FUNCTION_BLOCK FB_BaseControlElementDecoratorParent EXTENDS FB_BaseComponentDecoratorParent IMPLEMENTS ITF_BaseControlElementDecoratorParent
VAR
	itfControlElement				: ITF_BaseControlElement;
END_VAR

(*			
	EVERDE sp. z o.o.
	Rafał Osajda		24.03.2025		TC 4024.66
	Definicja nowego zgłoszenia
*)
METHOD PUBLIC EventsDefinition : BOOL
EventsDefinition		:= THIS^.itfControlElement.EventsDefinition ();
END_METHOD

(*			
	EVERDE sp. z o.o.
	Rafał Osajda		27.03.2025		TC 4024.66
	Obsluga bledow sprawdzanie czy jakis blad sie nei pojawil i ustawienie stanu lub wylaczenie
*)
METHOD PUBLIC ExecuteEveryCycle_Error
VAR_INPUT
END_VAR
THIS^.itfControlElement.ExecuteEveryCycle_Error ();
END_METHOD

(*			
	EVERDE sp. z o.o.
	Rafał Osajda		27.03.2025		TC 4024.66
	Wywolanie co cykl operacji 
*)
METHOD PUBLIC ExecuteEveryCycle_Operation
VAR_INPUT
END_VAR
THIS^.itfControlElement.ExecuteEveryCycle_Operation ();
END_METHOD

(*			
	EVERDE sp. z o.o.
	Rafał Osajda		27.03.2025		TC 4024.66
	Aktualizacja flag 
*)
METHOD PUBLIC ExecuteEveryCycle_Status
VAR_INST
END_VAR
THIS^.itfControlElement.ExecuteEveryCycle_Status ();
END_METHOD

(*			
	EVERDE sp. z o.o.
	Rafał Osajda		27.03.2025		TC 4024.66
	Testowanie czy nei pojawil sie jakis rozkaz i uruchomienie odpowiednich operacji
*)
METHOD PUBLIC ExecuteEveryCycle_Test
VAR_INPUT
END_VAR
THIS^.itfControlElement.ExecuteEveryCycle_Test ();
END_METHOD

METHOD FB_init : BOOL
VAR_INPUT
	bInitRetains : BOOL; // if TRUE, the retain variables are initialized (warm start / cold start)
	bInCopyCode : BOOL;  // if TRUE, the instance afterwards gets moved into the copy code (online change)
	fbToDecorate		: ITF_DecoratedElement;
END_VAR
THIS^.itfControlElement	:= fbToDecorate.GetITFControlElement ();
END_METHOD

(*			
	EVERDE sp. z o.o.
	Rafał Osajda		03.10.2025		TC 4024.66
	
*)
METHOD PUBLIC FirstCycle : BOOL
VAR_INPUT
END_VAR
FirstCycle				:= THIS^.itfControlElement.FirstCycle ();
END_METHOD

METHOD PUBLIC GetCode : STRING
VAR_INPUT
END_VAR
GetCode			:= THIS^.itfControlElement.GetCode ();
END_METHOD

(*			
	EVERDE sp. z o.o.
	Rafał Osajda		30.04.2025		TC 4024.66
	Zwraca czy element jest czymś zajety
*)
METHOD PUBLIC GetDoNothing : BOOL
GetDoNothing		:= THIS^.itfControlElement.GetDoNothing ();
END_METHOD

METHOD PUBLIC GetID : UINT
VAR_INPUT
END_VAR
GetID		:= THIS^.itfControlElement.GetID ();
END_METHOD

METHOD PUBLIC GetIdentyfier : ST_BaseElementIdentifier
VAR_INPUT
END_VAR
GetIdentyfier		:= THIS^.itfControlElement.GetIdentyfier ();
END_METHOD

METHOD PUBLIC GetName : ST_BaseLabel
VAR_INPUT
END_VAR
GetName		:= THIS^.itfControlElement.GetName ();
END_METHOD

(*			
	EVERDE sp. z o.o.
	Rafał Osajda		30.04.2025		TC 4024.66
	Zwraca czy element jest w pozycji 0 - referencyjnej
*)
METHOD PUBLIC GetPosition0 : BOOL
GetPosition0	:= THIS^.itfControlElement.GetPosition0 ();
END_METHOD

METHOD PUBLIC GetType : E_BaseElementType
VAR_INPUT
END_VAR
GetType		:= THIS^.itfControlElement.GetType ();
END_METHOD

(*			
	EVERDE sp. z o.o.
	Rafał Osajda		31.03.2025		TC 4024.66
	Flaga że w tej sesji pracy maszyny element został już wybazowany
*)
METHOD PUBLIC HomingGetDone : BOOL
VAR_INPUT
END_VAR
HomingGetDone	:= THIS^.itfControlElement.HomingGetDone ();
END_METHOD

(*			
	EVERDE sp. z o.o.
	Rafał Osajda		11.04.2025		TC 4024.66
	Zwraca czy bazowanie jest potrzebne
*)
METHOD PUBLIC HomingGetIsNeeded : BOOL
VAR_INPUT
END_VAR
HomingGetIsNeeded	:= THIS^.itfControlElement.HomingGetIsNeeded ();
END_METHOD

(*			
	EVERDE sp. z o.o.
	Rafał Osajda		27.05.2025		TC 4024.66
	Uruchomienie metody bazowania
*)
METHOD PUBLIC HomingStart
VAR_INPUT
END_VAR
THIS^.itfControlElement.HomingStart ();
END_METHOD

METHOD PUBLIC IsValidCommonData : BOOL
VAR_INPUT
END_VAR
IsValidCommonData			:= THIS^.itfControlElement.IsValidCommonData ();
END_METHOD

(*			
	EVERDE sp. z o.o.
	Rafał Osajda		07.10.2025		TC 4024.66
	Dodpisywanie się do listy logera
*)
METHOD PUBLIC JoinTheLogger : BOOL
VAR_INPUT
END_VAR
JoinTheLogger	:= THIS^.itfControlElement.JoinTheLogger ();
END_METHOD

METHOD PUBLIC LinkCommonData : BOOL
VAR_INPUT
	stCommonData				: REFERENCE TO ST_BaseCommonData;
END_VAR
LinkCommonData			:= THIS^.itfControlElement.LinkCommonData (stCommonData := stCommonData);
END_METHOD

METHOD PUBLIC LinkSS1 : BOOL
VAR_INPUT
	fbSS1			: ITF_BaseFlagGet;
END_VAR
LinkSS1		:= THIS^.itfControlElement.LinkSS1 (fbSS1 := fbSS1);
END_METHOD

METHOD PUBLIC LinkSTO : BOOL
VAR_INPUT
	fbSTO			: ITF_BaseFlagGet;
END_VAR
LinkSTO		:= THIS^.itfControlElement.LinkSTO (fbSTO := fbSTO);
END_METHOD

(*			
	EVERDE sp. z o.o.
	Rafał Osajda		31.03.2025		TC 4024.66
	Zwraca status zasilania	
*)
METHOD PUBLIC PowerGetStatus : BOOL
VAR_INPUT
END_VAR
PowerGetStatus		:= THIS^.itfControlElement.PowerGetStatus ();
END_METHOD

(*			
	EVERDE sp. z o.o.
	Rafał Osajda		31.03.2025		TC 4024.66
	Wyłączenie zasilania
*)
METHOD PUBLIC PowerTurnOff : BOOL
VAR_INPUT
END_VAR
PowerTurnOff		:= THIS^.itfControlElement.PowerTurnOff ();
END_METHOD

(*			
	EVERDE sp. z o.o.
	Rafał Osajda		31.03.2025		TC 4024.66
	Uruchomienie zasialania
*)
METHOD PUBLIC PowerTurnOn
VAR_INPUT
END_VAR
THIS^.itfControlElement.PowerTurnOn ();
END_METHOD

METHOD PUBLIC Reset : BOOL
VAR_INPUT
END_VAR
Reset	:= THIS^.itfControlElement.Reset ();
END_METHOD

METHOD PUBLIC ResetGetBusy : BOOL
VAR_INPUT
END_VAR
ResetGetBusy		:= THIS^.itfControlElement.ResetGetBusy ();
END_METHOD

METHOD PUBLIC ResetGetStatus : BOOL
VAR_INPUT
END_VAR
ResetGetStatus			:= THIS^.itfControlElement.ResetGetStatus ();
END_METHOD

METHOD PUBLIC SetCode
VAR_INPUT
	sCode							: STRING;
	sAdd							: STRING;
END_VAR
THIS^.itfControlElement.SetCode (sCode := sCode, sAdd := sAdd);
END_METHOD

(*			
	EVERDE sp. z o.o.
	Rafał Osajda		03.10.2025		TC 4024.66
	nadawanie unikalnych ID dla zdarzeń
*)
METHOD PUBLIC SetEventsIDs : UINT
VAR_INPUT
	uiNewID		: UINT;
END_VAR
SetEventsIDs		:= THIS^.itfControlElement.SetEventsIDs (uiNewID := uiNewID);
END_METHOD

METHOD PUBLIC SetID : UINT
VAR_INPUT
	uiID					: UINT;
END_VAR
SetID		:= THIS^.itfControlElement.SetID (uiID := uiID);
END_METHOD

METHOD PUBLIC SetName
VAR_INPUT
	stName				: ST_BaseLabel;
END_VAR
THIS^.itfControlElement.SetName (stName := stName);
END_METHOD

METHOD PUBLIC SetType
VAR_INPUT
	eType					: E_BaseElementType;
END_VAR
THIS^.itfControlElement.SetType (eType := eType);
END_METHOD

END_FUNCTION_BLOCK

(* stored: Version 1.1.0.1
   POU FB_BaseControlElementDecoratorParent: Id {b64f736c-95b6-0d2c-320a-88514714764e}, SpecialFunc None
   Folder Bazowanie: Id {84903104-6082-0efd-25eb-e2d7ce2bdbb4}
   Folder Events: Id {e9410f8a-e1db-054a-071b-fa572a90b062}
   Folder ID: Id {3efac1bf-e61b-0cd5-1379-2d160bc022c2}
   Folder ITF_BaseComponent: Id {e3476eae-0a1c-0790-23c5-ce328249c0e8}
   Folder WiazanieZmiennych: Id {d20cf12a-777b-0392-2614-f810b8f18269}
   Folder Zasilanie: Id {bedfc0d7-cf63-0e9f-2dfb-f19d9a8e3473}
   Method EventsDefinition: Id {972653cd-4023-08db-3afd-b91a624a9939}
   Method ExecuteEveryCycle_Error: Id {8eff9b7d-e6fc-04c1-3237-b231eff657ad}
   Method ExecuteEveryCycle_Operation: Id {0cf5555d-de63-0b69-2a2c-942019b00c0d}
   Method ExecuteEveryCycle_Status: Id {6910ee4c-2b65-0b52-2c89-7941228765d3}
   Method ExecuteEveryCycle_Test: Id {2f3b68c8-b242-0efe-2331-5d106f648809}
   Method FB_init: Id {69b9e0f4-87ec-069f-2ff7-9a4663046ec5}
   Method FirstCycle: Id {ac94cb0a-9636-0840-1b4b-ac78ca2533be}
   Method GetCode: Id {f8f9b47f-89a0-07f7-24d9-bd7a4f5a1618}
   Method GetDoNothing: Id {1375d626-888a-0f24-3cdc-5efde640af58}
   Method GetID: Id {8c7845f7-9cc5-006a-2d5a-2fd88072a75a}
   Method GetIdentyfier: Id {7076fce0-10f0-0357-35c1-ba97b1f217b0}
   Method GetName: Id {ec0ffe5c-f3a5-0070-17df-684ed4b488d4}
   Method GetPosition0: Id {a869147d-025c-0666-1100-ba9c5290550a}
   Method GetType: Id {6568029f-ec0b-0918-374d-2e0c3d4cf795}
   Method HomingGetDone: Id {114dd3ff-8c12-0211-179c-cacff92783c2}
   Method HomingGetIsNeeded: Id {433ac672-8ea7-0b59-3155-7a62393eae40}
   Method HomingStart: Id {a1094c07-d4bf-0a22-2255-bf1f37ebe64b}
   Method IsValidCommonData: Id {bf8382e8-3362-0a48-255b-3e609fe8b4eb}
   Method JoinTheLogger: Id {d99d488d-7f0f-078f-2ead-b83833883cf8}
   Method LinkCommonData: Id {3fe98781-29a8-0f0b-337b-84ae9e5d55d3}
   Method LinkSS1: Id {37a117fb-2f65-01f5-01bd-fd35ee4beb7f}
   Method LinkSTO: Id {43a829bd-758b-04cd-33a4-fa62ffad0f15}
   Method PowerGetStatus: Id {daf71b09-388d-0bf4-33ec-50043c4b8824}
   Method PowerTurnOff: Id {2f104ee1-676c-0c60-2492-e17661579837}
   Method PowerTurnOn: Id {48118c29-49fd-0d1f-1940-0850d6e694ee}
   Method Reset: Id {30c5b9ba-0aff-06a4-1542-82edd849d6a4}
   Method ResetGetBusy: Id {811cee6a-8edc-009c-310d-557d8d150a98}
   Method ResetGetStatus: Id {aca68a90-9aca-0775-1235-8f81b0e64507}
   Method SetCode: Id {947f1944-e673-0f09-0862-7cc193629ac4}
   Method SetEventsIDs: Id {962a51ed-714c-0571-33ae-4aa218f98eb4}
   Method SetID: Id {91d1b19e-a580-0afe-31b4-3ad2033d7039}
   Method SetName: Id {5a675704-2349-0e90-0793-792c7658a6b0}
   Method SetType: Id {0007d834-0427-0710-222e-6380b78ff489} *)
